// TIA Portal V19 export
TYPE "C501_VAR_NME_TYPIC"
   STRUCT
      MWA { ExternalAccessible := 'False'; ExternalVisible := 'False'; ExternalWritable := 'False'} : Real;   // Meetwaarde
      STS_HW { ExternalAccessible := 'False'; ExternalVisible := 'False'; ExternalWritable := 'False'} : USInt;   // Hoogwater vlotter
      STS_VHW { ExternalAccessible := 'False'; ExternalVisible := 'False'; ExternalWritable := 'False'} : USInt;   // Voorwaarschuwing hoogwater
      STS_SD { ExternalAccessible := 'False'; ExternalVisible := 'False'; ExternalWritable := 'False'} : USInt;   // Suppletie dicht
      STS_SO { ExternalAccessible := 'False'; ExternalVisible := 'False'; ExternalWritable := 'False'} : USInt;   // Suppletie open
      STS_VRL { ExternalAccessible := 'False'; ExternalVisible := 'False'; ExternalWritable := 'False'} : USInt;   // Voorwaarschuwing reservoir leeg
      STS_RL { ExternalAccessible := 'False'; ExternalVisible := 'False'; ExternalWritable := 'False'} : USInt;   // Reservoir leeg
      OBS { ExternalAccessible := 'False'; ExternalVisible := 'False'; ExternalWritable := 'False'} : USInt;   // Observeerbaarheid
   END_STRUCT;
END_TYPE
